{attribute 'GeneratedUsingTerminal: EK1960-0000-0019'}
{attribute addProperty BoxType "EK1960-0000-0019"}
{attribute addProperty Id "FSOEAT %I*FSOE_BBDEEE9E47"}
{attribute addProperty CRC "2458123369"}
{attribute addProperty Size "47"}
TYPE FSoE_Inputs_9283FC69 :
STRUCT
	{attribute addProperty Name "FSOE"}
	FSOE AT %I* : FSOE_BBDEEE9E;
END_STRUCT
END_TYPE

(* stored: Version 1.2.0.0, ProductVersion 3.1.4024.9
   DUT FSoE_Inputs_9283FC69: Id {4147a971-9c4b-4c24-9f15-f610d652dfae} *)
